TYPE ST_NestStatistics :
STRUCT
    uiNestId       : UINT;
    udiTotalTests  : UDINT;
    udiGoodParts   : UDINT;
    udiBadParts    : UDINT;
    lrEfficiency   : LREAL;
END_STRUCT
END_TYPE

(* stored: Version 1.1.0.1, ProductVersion 3.1.4026.18
   DUT ST_NestStatistics: Id {2ebb60dc-1705-4cd9-8d21-a2417fe407a4} *)
